TYPE ST_RelativeMovement :
STRUCT
END_STRUCT
END_TYPE

(* stored: Version 1.1.0.1, ProductVersion 3.1.4024.10
   DUT ST_RelativeMovement: Id {041cadc1-e239-404a-bbe6-a0a7d67ba383} *)
